Staubli VAL3: start.pgx

program start()
begin
   userPage(sEcran)
  cls(sEcran)
   putln(sEcran, "Quel programme voulez vous lancer : ")
  putln(sEcran, "   1. Découpe")
  putln(sEcran, "   2. Tour de 4 pièces")
  putln(sEcran, "   3. Constuire tour")
  get(sEcran, nYN)
  if nYN == 1
    call test_decoupe()
  elseIf nYN==2
    call saisirpiecev1()
  elseIf nYN==3
    call Tour()
  endIf
end
